{attribute addProperty BoxType "EK1122-0000-0018"}
{attribute addProperty Id "Beckhoff_ER1xxxsub_EK1100EK1100_179A0949162A_0001_ER1008_0001_0016ER1008_772BB4148210.25A_0002_ER1008_0001_0018ER1008_772BB4148210.25A_0003_ER1008_0002_0018ER1008_772BB4148210.25A_0004_ER1008_0022_0017ER1008_772BB4148210.25A_0005_ER1018_0001_0018ER1018_772BB4148210.25A_0006_ER1018_0002_0018ER1018_772BB4148210.25A_0007_ER1098_0001_0017ER1098_772BB4148210.25A_0008_ER1258_0001_0019ER1258_BB8E9A1042052.5A_0009_ER1258_0001_0020ER1258_BB8E9A1042052.5A_0010_ER1258_0002_0019ER1258_BB8E9A1042052.5A_0011_ER1258_0002_0020ER1258_BB8E9A1042052.5A_0012_ER1518_0002_0018ER1518_1EB154A835444.25A_0013_ER1518_0002_0019ER1518_1EB154A835444.25A_0014_ER1809_0021_0017ER1809_248EAA3414618.25A_0015_ER1809_0022_0018ER1809_248EAA3414618.25A_0016_ER1819_0021_0017ER1819_248EAA3414618.25A_0017_ER1819_0022_0017ER1819_248EAA3414618.25"}
{attribute addProperty CRC "62027282"}
{attribute addProperty SizeInBites "3562"}
{attribute addProperty SizeInBytes "445.25"}
TYPE Beckhoff_ER1xxxEK1122_03B27612 EXTENDS EK1122_179A0949 :
STRUCT
	{attribute addProperty Name "Beckhoff_ER1xxxsub_EK1100"}
	Beckhoff_ER1xxxsub_EK1100 : EK1100_179A0949;
	{attribute addProperty Name "A_0001_ER1008_0001_0016"}
	A_0001_ER1008_0001_0016 : ER1008_772BB414;
	{attribute addProperty Name "A_0002_ER1008_0001_0018"}
	A_0002_ER1008_0001_0018 : ER1008_772BB414;
	{attribute addProperty Name "A_0003_ER1008_0002_0018"}
	A_0003_ER1008_0002_0018 : ER1008_772BB414;
	{attribute addProperty Name "A_0004_ER1008_0022_0017"}
	A_0004_ER1008_0022_0017 : ER1008_772BB414;
	{attribute addProperty Name "A_0005_ER1018_0001_0018"}
	A_0005_ER1018_0001_0018 : ER1018_772BB414;
	{attribute addProperty Name "A_0006_ER1018_0002_0018"}
	A_0006_ER1018_0002_0018 : ER1018_772BB414;
	{attribute addProperty Name "A_0007_ER1098_0001_0017"}
	A_0007_ER1098_0001_0017 : ER1098_772BB414;
	{attribute addProperty Name "A_0008_ER1258_0001_0019"}
	A_0008_ER1258_0001_0019 : ER1258_BB8E9A10;
	{attribute addProperty Name "A_0009_ER1258_0001_0020"}
	A_0009_ER1258_0001_0020 : ER1258_BB8E9A10;
	{attribute addProperty Name "A_0010_ER1258_0002_0019"}
	A_0010_ER1258_0002_0019 : ER1258_BB8E9A10;
	{attribute addProperty Name "A_0011_ER1258_0002_0020"}
	A_0011_ER1258_0002_0020 : ER1258_BB8E9A10;
	{attribute addProperty Name "A_0012_ER1518_0002_0018"}
	A_0012_ER1518_0002_0018 : ER1518_1EB154A8;
	{attribute addProperty Name "A_0013_ER1518_0002_0019"}
	A_0013_ER1518_0002_0019 : ER1518_1EB154A8;
	{attribute addProperty Name "A_0014_ER1809_0021_0017"}
	A_0014_ER1809_0021_0017 : ER1809_248EAA34;
	{attribute addProperty Name "A_0015_ER1809_0022_0018"}
	A_0015_ER1809_0022_0018 : ER1809_248EAA34;
	{attribute addProperty Name "A_0016_ER1819_0021_0017"}
	A_0016_ER1819_0021_0017 : ER1819_248EAA34;
	{attribute addProperty Name "A_0017_ER1819_0022_0017"}
	A_0017_ER1819_0022_0017 : ER1819_248EAA34;
END_STRUCT
END_TYPE

(* stored: Version 1.2.0.0, ProductVersion 3.1.4024.9
   DUT Beckhoff_ER1xxxEK1122_03B27612: Id {e2d03602-e54c-4bc8-b27f-c97b19e1db21} *)
